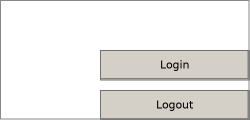
VISUALIZATION VISU_TEST_LOGIN  // 250x120
    Button (100,50 150x30), "Login"
        OnMouseDown: VisuUserMgmt Type=Login
    Button (100,90 150x30), "Logout"
        OnMouseDown: VisuUserMgmt Type=Logout
END_VISUALIZATION

(* stored: Version 1.1.0.1, ProductVersion 3.1.4024.11
   Visu VISU_TEST_LOGIN: Id {af83bbf7-4634-47a5-8b47-8c8d94650187} *)
